TYPE ST_EstoqueSnapshot :
STRUCT
	nA : INT;
	nB : INT;
	nC : INT;
END_STRUCT
END_TYPE

(* stored: Version 1.1.0.1
   DUT ST_EstoqueSnapshot: Id {951d7b35-af37-4295-876b-ab9d164883ac} *)
